TYPE EtcSlaveBase_82538BE2 : 
STRUCT
END_STRUCT
END_TYPE

(* stored: Version 1.1.0.1, ProductVersion 3.1.4024.9
   DUT EtcSlaveBase_82538BE2: Id {f846f1fc-68e6-0bd7-19bc-8072382496ee} *)
